TYPE
    GeneralDeviceInformation :
    STRUCT
        DeviceType      : UDINT;
        DeviceName      : STRING;
        HardwareVersion : STRING;
        SoftwareVersion : STRING;
    END_STRUCT
END_TYPE

(* stored: Version 1.1.0.1, ProductVersion 3.1.4024.12
   DUT GeneralDeviceInformation: Id {e7e106f0-9e49-0bcd-21d3-7759971c6903} *)
